// TIA Portal V19 export
DATA_BLOCK "DB_Exchange"   // DB1
{ S7_Optimized_Access := 'TRUE'; DB_Accessible_From_OPC_UA := 'FALSE' }
// stored: AutoNumber false, DBAccessibleFromOPCUA false, DBAccessibleFromWebserver false, MemoryReserve 100
   VAR
      xAutoMode { ExternalAccessible := 'False'; ExternalVisible := 'False'; ExternalWritable := 'False'} : Bool;   // Automatic mode
      xSemiAutoMode { ExternalAccessible := 'False'; ExternalVisible := 'False'; ExternalWritable := 'False'} : Bool;   // Semi-automatic mode
      xMaintenanceMode { ExternalAccessible := 'False'; ExternalVisible := 'False'; ExternalWritable := 'False'} : Bool;   // Maintenance mode
      xAuthorizationStartSanding { ExternalAccessible := 'False'; ExternalVisible := 'False'; ExternalWritable := 'False'} : Bool;
      xLeftRobotStartVacuum { ExternalAccessible := 'False'; ExternalVisible := 'False'; ExternalWritable := 'False'} : Bool;   // Left Robot request start vacuum
      xRightRobotStartVacuum { ExternalAccessible := 'False'; ExternalVisible := 'False'; ExternalWritable := 'False'} : Bool;   // Right Robot request start vacuum
      xStopRobotRequested { ExternalAccessible := 'False'; ExternalVisible := 'False'; ExternalWritable := 'False'} : Bool;   // Stop robot requested for openning the door
      xLeftRobotStopped { ExternalAccessible := 'False'; ExternalVisible := 'False'; ExternalWritable := 'False'} : Bool;   // Left Robot stopped in good position
      xRightRobotStopped { ExternalAccessible := 'False'; ExternalVisible := 'False'; ExternalWritable := 'False'} : Bool;   // Right Robot stopped in good position
      xGlobalFault { ExternalAccessible := 'False'; ExternalVisible := 'False'; ExternalWritable := 'False'} : Bool;   // Cell Global Fault
      xGlobalWarning { ExternalAccessible := 'False'; ExternalVisible := 'False'; ExternalWritable := 'False'} : Bool;   // Cell Global warning
      xInformation { ExternalAccessible := 'False'; ExternalVisible := 'False'; ExternalWritable := 'False'} : Bool;   // An information message is display
      xConditionOk { ExternalAccessible := 'False'; ExternalVisible := 'False'; ExternalWritable := 'False'} : Bool;   // Condition to run ok
      xStartUpWarningLeft { ExternalAccessible := 'False'; ExternalVisible := 'False'; ExternalWritable := 'False'} : Bool;   // Start up warning before left robot run
      xStartUpWarningRight { ExternalAccessible := 'False'; ExternalVisible := 'False'; ExternalWritable := 'False'} : Bool;   // Start up warning before right robot run
      xReqOperatorAction { ExternalAccessible := 'False'; ExternalVisible := 'False'; ExternalWritable := 'False'} : Bool;   // Request operator action
      xRecipeOpeInProgress { ExternalAccessible := 'False'; ExternalVisible := 'False'; ExternalWritable := 'False'} : Bool;   // Recipe Operation in progress
      xSandingInProgress { ExternalAccessible := 'False'; ExternalVisible := 'False'; ExternalWritable := 'False'} : Bool;   // Sanding process is in progress
      xUnloadRecipe { ExternalAccessible := 'False'; ExternalVisible := 'False'; ExternalWritable := 'False'} : Bool;   // Unload current recipe
      xProductionRunningRobot1 { ExternalAccessible := 'False'; ExternalVisible := 'False'; ExternalWritable := 'False'} : Bool;   // Production running on Robot 1
      xProductionRunningRobot2 { ExternalAccessible := 'False'; ExternalVisible := 'False'; ExternalWritable := 'False'} : Bool;   // Production running on Robot 2
      xStartSanding { ExternalAccessible := 'False'; ExternalVisible := 'False'; ExternalWritable := 'False'} : Bool;   // Beginning of sanding
      xEndSanding { ExternalAccessible := 'False'; ExternalVisible := 'False'; ExternalWritable := 'False'} : Bool;   // End of sanding
      udiVacuumRunningTime { ExternalAccessible := 'False'; ExternalVisible := 'False'; ExternalWritable := 'False'} : UDInt;   // Vacuum Running time
      LeftRobot { ExternalAccessible := 'False'; ExternalVisible := 'False'; ExternalWritable := 'False'} : Struct
         udiFaultTime : UDInt;
         udiRunTime : UDInt;
         udiPauseTime : UDInt;
         udiRobotPowerOnTime : UDInt;
         udiRobotDriveOnTime : UDInt;
         xRobotUsed : Bool;
      END_STRUCT;
      RightRobot { ExternalAccessible := 'False'; ExternalVisible := 'False'; ExternalWritable := 'False'} : Struct
         udiFaultTime : UDInt;
         udiRunTime : UDInt;
         udiPauseTime : UDInt;
         udiRobotPowerOnTime : UDInt;
         udiRobotDriveOnTime : UDInt;
         xRobotUsed : Bool;
      END_STRUCT;
      stLeftRobotFlatnessCtrlData { ExternalAccessible := 'False'; ExternalVisible := 'False'; ExternalWritable := 'False'} : "stFlatnessData";
      stRightRobotFlatnessCtrlData { ExternalAccessible := 'False'; ExternalVisible := 'False'; ExternalWritable := 'False'} : "stFlatnessData";
   END_VAR
BEGIN
END_DATA_BLOCK
